Fanuc TP program (LS listing): chwytak1.ls

/PROG  CHWYTAK1	  Macro
/ATTR
OWNER		= MNEDITOR;
COMMENT		= "";
PROG_SIZE	= 152;
CREATE		= DATE 17-02-06  TIME 09:09:18;
MODIFIED	= DATE 17-02-06  TIME 09:45:20;
FILE_NAME	= ;
VERSION		= 0;
LINE_COUNT	= 1;
MEMORY_SIZE	= 520;
PROTECT		= READ_WRITE;
TCD:  STACK_SIZE	= 0,
      TASK_PRIORITY	= 50,
      TIME_SLICE	= 0,
      BUSY_LAMP_OFF	= 0,
      ABORT_REQUEST	= 0,
      PAUSE_REQUEST	= 0;
DEFAULT_GROUP	= *,*,*,*,*;
CONTROL_CODE	= 00000000 00000000;
/APPL
/MN
   1:  RO[1:otworz chwytak 1]=(!RO[1:otworz chwytak 1]) ;
/POS
/END
